PROGRAM P11_E3508
VAR
	wControlValue			: WORD;
	wPowerRateSetValue		: WORD;	
	bOutputManAuto 			: BOOL; // Command 0:Auto, 1:Manual Mode
	
	bHeaterOn				: BOOL := FALSE; //to PSTEK
	bHeaterReset			: BOOL; //to PSTEK

	bAlarmState_E3508 		: BOOL; //Alarm or Sensor Break Signal
	bManAuto_E3508 			: BOOL; //State, 0:Manual, 1:Auto

	isHeaterReady			: BOOL; //Close : Ready
	isHeaterRun				: BOOL; //Close : Running, Open : Stop
	isHeaterFault			: BOOL; //Close : Falut, Open : Normal
	//isInductionHeaterErr	: BOOL; //Power Supply
	bInductionHeaterCB		: BOOL;
	//Input from E3508 Controller
	aInputPVBytes AT %I* 		: ARRAY[1..2]OF USINT; //Input Process Values
	aInputSVBytes AT %I* 		: ARRAY[1..2]OF USINT; //Input Set Values
	aInputTVBytes AT %I* 		: ARRAY[1..2]OF USINT; //Input Target Valuse
	aInputCVBytes AT %I* 		: ARRAY[1..2]OF USINT; //Induction Heter Controlled Values
	aInputProportional AT %I* 	: ARRAY[1..2]OF USINT; //PID - Proportional Band
	aInputIntegral AT %I* 		: ARRAY[1..2]OF USINT; //PID - Integral Time
	aInputDerivative AT %I* 	: ARRAY[1..2]OF USINT; //PID - Derivative Time 
	nInputAlarmBytes AT %I* 	: USINT; // Alarm State
	nInputManAutoBytes AT %I* 	: USINT; // ManAuto State
	
	wE3508_PV				: WORD;
	wE3508_SV				: WORD;
	wE3508_PowerRate		: WORD; //To Induction Heater Control Values
	wE3508_P				: WORD; //PID Parameter P
	wE3508_I				: WORD; //PID Parameter I
	wE3508_D				: WORD; //PID Parameter D
	//Output to E3508 Controller
	wOutputSVBytes 				: outWord;
	wOutputPowerSVBytes 		: outWord;
	aOutputSVBytes AT %Q* 		: ARRAY[1..2]OF USINT; //Temperature Set Value
	nOutputManAutoBytes AT %Q* 	: USINT; //ManAuto Change
	aOutputPowerBytes AT %Q* 	: ARRAY[1..2]OF USINT; //Output Power in Manual State
	//nOutputAlarmClear AT %Q* : USINT; //Alarm Clear Set
END_VAR

//Induction Heater & Temperature Controller & Thermo Couple(R-Type)
//Maker: PSTEK, Eurotherm
//Model: 3508
//Temperature Range: 0 ~ 12000℃

(* Command *)
bHeaterOn := GVL_IO.aOutputCmd[1].4;
bHeaterReset := GVL_IO.aOutputCmd[1].5;
nOutputManAutoBytes.0 := GVL_IO.aOutputCmd[1].11; //Temp Controller Mode Command

(* Read from Power Distribution Pannel *)
bInductionHeaterCB		:= GVL_IO.aDigitalInputIO[4].7;
nInputAlarmBytes.7 		:= GVL_IO.aInputState[4].7;
nInputManAutoBytes.7 	:= GVL_IO.aInputState[4].8;

(* Read from E3508 Device Value *)
wE3508_PV				:= USINT_TO_WORD_Bit(aInputPVBytes[1], aInputPVBytes[2]);
wE3508_SV				:= USINT_TO_WORD_Bit(aInputSVBytes[1], aInputSVBytes[2]);
wE3508_PowerRate		:= USINT_TO_WORD_Bit(aInputCVBytes[1], aInputCVBytes[2]); //divided to 10
wE3508_P 				:= USINT_TO_WORD_Bit(aInputProportional[1], aInputProportional[2]);
wE3508_I 				:= USINT_TO_WORD_Bit(aInputIntegral[1], aInputIntegral[2]);
wE3508_D 				:= USINT_TO_WORD_Bit(aInputDerivative[1], aInputDerivative[2]);

//bAlarmState_E3508 		:= nInputAlarmBytes.7;

GVL_IO.aMonitoring_PV[10] := WORD_TO_REAL(wE3508_PowerRate)*0.1; //divided to 10 PowerRate

(* Read from Induction Heater Value *)
isHeaterReady 			:= GVL_IO.aDigitalInputIO[2].2;
isHeaterRun		 		:= GVL_IO.aDigitalInputIO[2].3;
isHeaterFault 			:= GVL_IO.aDigitalInputIO[2].4;

// Interface with other PRGs
wControlValue			:= LREAL_TO_WORD(GVL_IO.aController[27].rControlValue);
GVL_IO.wE3508_PV		:= wE3508_PV;

(* Write to E3508 Device Value *)
// Operation Mode
// bOutputManAuto := GVL_IO.aOutputCmd[1].11; //Temp Controller Mode Command
// nOutputManAutoBytes.0 	:= GVL_IO.aOutputCmd[1].11; //Command

IF nInputManAutoBytes.7 THEN // Read form E3508 Mode, 0:Man 1:Auto
	wOutputPowerSVBytes 	:= WORD_TO_USINT_Bit(wControlValue*10); //multiple to 10, Power Reate Set Value
	aOutputPowerBytes[1] 	:= wOutputPowerSVBytes.Lower;
	aOutputPowerBytes[2] 	:= wOutputPowerSVBytes.Upper;
ELSE
	wOutputSVBytes 			:= WORD_TO_USINT_Bit(wControlValue); // Temperature Set Value
	aOutputSVBytes[1] 		:= wOutputSVBytes.Lower;
	aOutputSVBytes[2] 		:= wOutputSVBytes.Upper;
END_IF

(* Write to Induction Heater Value *)
GVL_IO.aDigitalOutputIO[2].0 := bHeaterOn;
GVL_IO.aDigitalOutputIO[2].1 := bHeaterReset;
GVL_IO.nE3508_nInputManAutoBytes := nInputManAutoBytes; //State

END_PROGRAM

(* stored: Version 1.1.0.1, ProductVersion 3.1.4026.11
   POU P11_E3508: Id {a7e3d6a1-82f0-4607-8ac9-093cb5f931f5}, SpecialFunc None *)
